FUNCTION F_InitializeAllFunctions :BOOL
(**************************************************************************************
 * 	Application		:	BoxControl Framework
 *	Revision		:	$Revision: 404529 $
 *	Revision date	:	$Date: 2018-04-23 08:21:38 +0200 (Mo., 23 Apr 2018) $
 *	Last changed by	:	$Author: b7bolm $
 *	URL				:	$URL: http://almscdc.swisslog.com/repo/SWPD/Development/BoxControlFramework/20_Release/trunk/01_Software/BCF/BCF/JumpStart/20_Product/10_App/12_E_Functions/10_Lib/10_Conv/10_Functions/F_InitializeAllFunctions.TcPOU $
 *
 *	Purpose			:	Initialize all functions
 *
 * ------------------------------------------------------------------------------------
 *	Copyright Swisslog [IP AG], Switzerland. All rights reserved.
 * 
 * ------------------------------------------------------------------------------------
 *	
 * 	Revision History: 
 *
 * 	VERSION			DATE			INITIALS			DESCRIPTION
 *	0.1				01.01.2001		swl					Example
 *
 **************************************************************************************)
VAR
	eFunctionNumber		: E_FunctionNumber; // Function number

END_VAR

// Loop over all elements and initialize each function 
FOR eFunctionNumber := E_FunctionNumber.F_BEGIN_FUNCTION + 1 TO E_FunctionNumber.F_END_FUNCTION - 1 DO
	// If reference is valid
	IF __ISVALIDREF(FunctionRegistry[eFunctionNumber].rFunction) THEN
		// Initialize function
		FunctionRegistry[eFunctionNumber].rFunction.M_InitFunction(TRUE);
	END_IF
END_FOR

END_FUNCTION

(* stored: Version 1.1.0.1, ProductVersion 3.1.4022.12
   POU F_InitializeAllFunctions: Id {f5e8f4b4-a38f-4f86-949b-807ea192a4fd}, SpecialFunc None *)
